# B&R Automation Studio project DynamicIO
Automation Studio 4.5.2.102

## Configuration 5AP1120

CPU 5PC901.TS77-00, AutomationRuntime D4.52, Build 4.1.2, Vc V4.52.0

### Task classes (Cpu.sw)
```
Cyclic#4:
  XmlConfigT <- Logic.XmlConfigTest.prg
  AsIoMManTe <- Logic.AsIoMManTest.prg
  ModuleIden <- Logic.ModuleIdent.prg [disabled]
Binaries: udbdef, TCData, ashwac, arconfig, asfw, ashwd, iomap, User, Role, sysconf
Libraries: standard, AsIOMMan, runtime, DataObj, AsXml, FileIO
```

### Hardware
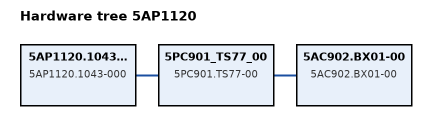
```
5AC902.BX01-00 : 5AC902.BX01-00 v1.1.1.0  [SY -> 5PC901_TS77_00.SY3]
5AP1120.1043-000 : 5AP1120.1043-000 v1.3.0.0
5PC901_TS77_00 : 5PC901.TS77-00 v2.0.0.0  [SY -> 5AP1120.1043-000.SY1]
  Connector IF1:
    AssignedOperatingSystem = ARemb
  Connector IF2:
    AssignedOperatingSystem = ARemb
  Connector IF3:
    AssignedOperatingSystem = ARemb
    ActivateDevice = 1
  Connector IF4:
    AssignedOperatingSystem = ARemb
    ActivateDevice = 1
  Connector IF5:
    AssignedOperatingSystem = ARemb
  Connector IF6:
    AssignedOperatingSystem = ARemb
  Connector IF7:
    AssignedOperatingSystem = ARemb
  Connector IF8:
    AssignedOperatingSystem = ARemb
  ConfigurationID = DynamicIO_5AP1120
  Simulation = 1
  FileDevice1
  FileDeviceName1 = root
  FileDevicePath1 = E:/
```

## Configuration CP3585

CPU X20CP3585, AutomationRuntime D4.52, Build 4.1.2, Vc V4.52.0

### Task classes (Cpu.sw)
```
Cyclic#3:
  XmlEditor <- Logic.XmlEditor.prg
Cyclic#4:
  IomapParse <- Logic.IomapParser.prg
  XmlConfigT <- Logic.XmlConfigTest.prg
  AsIoMManTe <- Logic.AsIoMManTest.prg
  ModuleIden <- Logic.ModuleIdent.prg
Binaries: udbdef, TCData, ashwac, arconfig, asfw, ashwd, iomap, User, Role, sysconf
Libraries: standard, AsIOMMan, runtime, DataObj, AsXml, FileIO, AsIODiag
```

### Hardware
```
X20BM11 : X20BM11 v1.0.0.1  [X2X1 -> X20CP3585.IF6]
X20CP3585 : X20CP3585 v1.5.0.0
  Connector IF2:
    ActivateDevice = 1
  ConfigurationID = DynamicIO_5AP1120
  Simulation = 1
  FileDevice1
  FileDeviceName1 = root
  FileDevicePath1 = E:/
X20DOF322 : X20DOF322 v1.1.2.0  [SS1 -> X20TB1F.SS; SL -> X20BM11.SL1]
X20TB1F : X20TB1F v1.0.0.0
```

## Logical view

Binary libraries used (declarations not repeated): operator, runtime, astime, AsIecCon, standard, AsIOMMan, DataObj, AsXml, FileIO, AsIODiag

### Global.typ - Global data types
```iecst
TYPE
	Module_type : 	STRUCT
		ModuleName : STRING[80];
		ModulePath : STRING[80];
		ChannelType : STRING[80] := 'BOOL';
		Channel : ARRAY[0..15]OF Channel_type;
		ModuleType : STRING[10] := '%QX';
	END_STRUCT;
	Channel_type : 	STRUCT
		ChannelVar : STRING[80];
		ChannelName : STRING[80];
	END_STRUCT;
END_TYPE
```

### Global.var - Global variables
```iecst
VAR
	X20DIF371 : Module_type;
	DI : ARRAY[0..15] OF BOOL;
	DigOut : ARRAY[0..15] OF BOOL;
	HW_config : Module_type;
	New_Variable : {REDUND_UNREPLICABLE} USINT := 4;
END_VAR
```


### Program Logical/Logic/ModuleIdent (ANSIC)

#### Types.typ
```iecst
TYPE
	ShowModules :
		(
		CONFIGURED_MODULES := 2,
		ALL := 3,
		PLUGGED := 1
		);
	ModuleInfo :
		(
		EPLAN_MODULE_TAG := 1007,
		HW_MODULE_NAME := 1006,
		PLUGGED_MODULE_BUS := 1004,
		CONFIGURATED_MODULE_BUS := 1005,
		PLUGGED_MODULE_NAME := 1002,
		CONFIG_MODULE_NAME := 1003,
		MODULE_PATH := 1001
		);
END_TYPE
```

#### Variables.var
```iecst
VAR
	GetInfo : DiagCreateInfo;
	Ident : UDINT;
	GetNumInfo : DiagGetNumInfo;
	GetStrInfo : DiagGetStrInfo;
	InfoDesc : STRING[80];
	start : BOOL;
	ConnectedModuleList : ARRAY[0..9] OF STRING[80];
	i : USINT;
END_VAR
```

#### Main.c
```c
#include <bur/plctypes.h>
#define TRUE	1
#define FALSE 	0

#ifdef _DEFAULT_INCLUDES
	#include <AsDefault.h>
#endif

void _INIT ProgramInit(void)
{

}

void _CYCLIC ProgramCyclic(void)
{
//	Тест опроса текущей конфигурации
	if(start)
	{
		if(GetInfo.ident == 0)	GetInfo.enable = TRUE;

		if(GetInfo.enable)
		{
			GetInfo.infoKind = CONFIGURED_MODULES;
			DiagCreateInfo(&GetInfo);
			Ident = GetInfo.ident;
			GetStrInfo.ident = Ident;
			GetStrInfo.enable = TRUE;
			GetStrInfo.infoCode = HW_MODULE_NAME;

			i = 0;
			if(GetInfo.status == 0)
			{
				GetInfo.enable = FALSE;
			}
		}
		if(	i < ( GetInfo.nrEntries) )
		{
			GetStrInfo.index = i;
			GetStrInfo.bufferLen = sizeof(InfoDesc);
			GetStrInfo.pBuffer = &InfoDesc;
			DiagGetStrInfo(&GetStrInfo);
			strcpy(ConnectedModuleList[GetStrInfo.index],InfoDesc);

			if(i == ( GetInfo.nrEntries - 1))
			{
				GetStrInfo.enable = FALSE;
				start = FALSE;
			}
			if(GetStrInfo.status == 0) i++;
		}
	}
}

void _EXIT ProgramExit(void)
{

}
```

### Program Logical/Logic/AsIoMManTest (ANSIC)

#### Types.typ
```iecst
TYPE
	FileMgrStep_enum :
		(
		CREATE,
		OPEN,
		WRITE,
		CLOSE
		);
	ReadCfg_enum :
		(
		Wait,
		CopyCfg,
		GetDatObjData,
		WriteXML
		);
END_TYPE
```

#### Variables.var
```iecst
VAR
	IOMMCopy : AsIOMMCopy;
	RemoveBr : AsIOMMRemove;
	CreateBr : AsIOMMCreate;
	status_message : STRING[128];
	error_string : STRING[128];
	step : USINT;
	error_status : UINT;
	error_step : USINT;
	error : BOOL;
	config : UINT;
	change_config : UINT;
	DataObjName : STRING[80];
	BR_ModuleName : STRING[80];
	DO_Create : DatObjCreate;
	DO_Read : DatObjRead;
	DO_Info : DatObjInfo;
	FileName : STRING[80];
	CfgReadStep : ReadCfg_enum;
	FW_Step : FileMgrStep_enum;
	Start : BOOL;
	fCreate : FileCreate;
	fOpen : FileOpen;
	fClose : FileClose;
	fRead : FileRead;
	fWrite : FileWrite;
	fIdent : UDINT;
END_VAR
```

#### Main.c
```c
#include <bur/plctypes.h>
#define	TRUE	1
#define	FALSE	0

#ifdef _DEFAULT_INCLUDES
	#include <AsDefault.h>
#endif

void _INIT ProgramInit(void)
{

}

void _CYCLIC ProgramCyclic(void)
{
	switch(CfgReadStep)
	{
		case Wait:
			if(Start)
			{
				CfgReadStep	= CopyCfg;
			}
			break;

		case CopyCfg:
			IOMMCopy.enable			= TRUE;
			IOMMCopy.pModuleName	= &BR_ModuleName;
			IOMMCopy.pNewModule		= &DataObjName;
			AsIOMMCopy(&IOMMCopy);
			if(IOMMCopy.status == ERR_OK)
			{
				CfgReadStep	= GetDatObjData;
			}
			break;

		case GetDatObjData:
			DO_Info.enable	= TRUE;
			DO_Info.pName	= IOMMCopy.pNewModule;
			DatObjInfo(&DO_Info);
			if(DO_Info.status == ERR_OK)
			{
				CfgReadStep	= WriteXML;
			}
			break;

		case WriteXML:
			switch (FW_Step)
			{

				case CREATE:
					fCreate.enable	= TRUE;
					fCreate.pDevice = (UDINT) "root";
					fCreate.pFile 	= &FileName;
					FileCreate(&fCreate);
					if(fCreate.status == ERR_OK)
					{
						fIdent	= fCreate.ident;
						FW_Step	= WRITE;
					}
					else if(fCreate.status == fiERR_EXIST)
					{
						FW_Step	= OPEN;
					}
					break;

				case OPEN:
					fOpen.pDevice	= (UDINT) "root";//= fCreate.pDevice;
					fOpen.pFile		= &FileName;//fCreate.pFile;
					fOpen.mode		= FILE_RW;
					fOpen.enable	= TRUE;
					FileOpen(&fOpen);
					if(fOpen.status == ERR_OK)
					{
						fIdent	= fOpen.ident;
						FW_Step	= WRITE;
					}
					break;

				case WRITE:
					fWrite.ident	= fIdent;
					fWrite.offset	= 0;
					fWrite.pSrc		= DO_Info.pDatObjMem;
					fWrite.len		= DO_Info.len;
					fWrite.enable	= TRUE;
					FileWrite(&fWrite);
					if(fWrite.status == ERR_OK)
					{
						FW_Step	= CLOSE;
					}
					break;

				case CLOSE:
					fClose.ident	= fIdent;
					fClose.enable	= TRUE;

					FileClose(&fClose);
					if(fClose.status == ERR_OK)
					{
						Start		= FALSE;
						CfgReadStep	= Wait;
					}
					break;

			}
	}
}

void _EXIT ProgramExit(void)
{

}
```

### Program Logical/Logic/XmlConfigTest (ANSIC)

#### Types.typ
```iecst
TYPE
	ProgramStep_enum :
		(
		Wait,
		WriteEndDoc,
		CreateMem,
		WriteArV,
		WriteHeader,
		WriteIO_Tag,
		WriteIO_TagAttr,
		WriteLinksTag,
		WriteLinkNodes,
		WriteLinksTagEnd,
		WriteIO_TagEnd,
		GetMemPointer,
		WriteDataObj,
		CopyXML,
		RemoveOldIomap,
		CreateNewIomap,
		DeleteDatObj,
		WarmRestart
		);
	FileMgrStep_enum :
		(
		CREATE,
		OPEN,
		WRITE,
		CLOSE
		);
	WriteLNStep_enum :
		(
		WriteLN_Tag,
		WriteLN_ID,
		WriteLN_Type,
		WriteProdTag,
		WriteProdDevice,
		WriteProdDPName,
		WriteProdKind,
		WriteProd_TagEnd,
		WriteConsTag,
		WriteConsDevice,
		WriteConsDPName,
		WriteConsKind,
		WriteCons_TagEnd,
		WriteLN_TagEnd
		);
	ModuleType : 	STRUCT
		ModuleName : STRING[80];
		ModulePath : STRING[80];
		ModuleType : STRING[80];
		ChanelNumber : USINT;
		ChanelType : STRING[80];
		ChanelVarName : ARRAY[0..15]OF STRING[80];
		ChanelName : ARRAY[0..15]OF STRING[80];
	END_STRUCT;
END_TYPE
```

#### Variables.var
```iecst
VAR
	CreateMemory : xmlCreateMemoryWriter;
	WriteStartDocument : xmlWriteStartDocument;
	WriteStartElement : xmlWriteStartElement;
	WriteAttribute : xmlWriteAttribute;
	WriteElementText : xmlWriteElementText;
	WriteEndElement : xmlWriteEndElement;
	WriteEndDocument : xmlWriteEndDocument;
	WritePI : xmlWritePI;
	GetMemoryInfo : xmlGetMemoryInfo;
	Step : ProgramStep_enum;
	Start : BOOL;
	XmlData : STRING[1000];
	Ident : UDINT;
	IO_AttrName : STRING[80] := 'xmlns';
	IOTagName : STRING[80] := 'IO';
	XmlEnc : STRING[80] := 'utf-8';
	fIdent : UDINT;
	XmlVer : STRING[80] := '1.0';
	IOAttrValue : STRING[80] := 'http://www.br-automation.com/AR/IO\';
	ArName : STRING[80] := 'AutomationRuntimeIOSystem';
	ArVer : STRING[80] := 'Version=\"1.0\"';
	fCreate : FileCreate;
	fOpen : FileOpen;
	fClose : FileClose;
	fRead : FileRead;
	LN_Step : WriteLNStep_enum;
	fWrite : FileWrite;
	FW_Step : FileMgrStep_enum;
	i : USINT := 5;
	DO_Delete : DatObjDelete;
	DO_Create : DatObjCreate;
	DO_Write : DatObjWrite;
	DO_Info : DatObjInfo;
	DataObj_Step : USINT;
	DOF322 : ModuleType;
	Buff : STRING[80];
	IOMMRemove : AsIOMMRemove;
	IOMMCreate : AsIOMMCreate;
END_VAR
```

#### Main.c
```c
#include <bur/plctypes.h>
#define TRUE	1
#define FALSE	0
UDINT StringCombiner(STRING* pDest,STRING* pIoType, STRING* pSrc1, STRING* pSrc2)
{
	strcpy(pDest,pIoType);
	strcat(pDest,".");
	strcat(pDest,pSrc1);
	strcat(pDest,".");
	strcat(pDest,pSrc2);
	return pDest;
}
#ifdef _DEFAULT_INCLUDES
	#include <AsDefault.h>
#endif

void _INIT ProgramInit(void)
{

	DigOut[1]	=	DigOut[1];
	DigOut[2]	=	DigOut[2];
	DigOut[3]	=	DigOut[3];
	DigOut[4]	=	DigOut[4];
	DigOut[5]	=	DigOut[5];
	DigOut[6]	=	DigOut[6];
	DigOut[7]	=	DigOut[7];
	DigOut[8]	=	DigOut[8];
	DigOut[9]	=	DigOut[9];
	DigOut[10]	=	DigOut[10];
	DigOut[11]	=	DigOut[11];
	DigOut[12]	=	DigOut[12];
	DigOut[13]	=	DigOut[13];
	DigOut[14]	=	DigOut[14];
	DigOut[15]	=	DigOut[15];

	Step	= Wait;
}

void _CYCLIC ProgramCyclic(void)
{
	switch(Step)
	{
		case Wait:
			if(Start)
			{
				strcpy(DOF322.ChanelName[0],"DigitalOutput01");
				strcpy(DOF322.ChanelName[1],"DigitalOutput02");
				strcpy(DOF322.ChanelName[2],"DigitalOutput03");
				strcpy(DOF322.ChanelName[3],"DigitalOutput04");
				strcpy(DOF322.ChanelName[4],"DigitalOutput05");
				strcpy(DOF322.ChanelName[5],"DigitalOutput06");
				strcpy(DOF322.ChanelName[6],"DigitalOutput07");
				strcpy(DOF322.ChanelName[7],"DigitalOutput08");
				strcpy(DOF322.ChanelName[8],"DigitalOutput09");
				strcpy(DOF322.ChanelName[9],"DigitalOutput10");
				strcpy(DOF322.ChanelName[10],"DigitalOutput11");
				strcpy(DOF322.ChanelName[11],"DigitalOutput12");
				strcpy(DOF322.ChanelName[12],"DigitalOutput13");
				strcpy(DOF322.ChanelName[13],"DigitalOutput14");
				strcpy(DOF322.ChanelName[14],"DigitalOutput15");
				strcpy(DOF322.ChanelName[15],"DigitalOutput16");

				strcpy(DOF322.ChanelVarName[0],"::DigOut[15]");
				strcpy(DOF322.ChanelVarName[1],"::DigOut[14]");
				strcpy(DOF322.ChanelVarName[2],"::DigOut[13]");
				strcpy(DOF322.ChanelVarName[3],"::DigOut[12]");
				strcpy(DOF322.ChanelVarName[4],"::DigOut[11]");
				strcpy(DOF322.ChanelVarName[5],"::DigOut[10]");
				strcpy(DOF322.ChanelVarName[6],"::DigOut[9]");
				strcpy(DOF322.ChanelVarName[7],"::DigOut[8]");
				strcpy(DOF322.ChanelVarName[8],"::DigOut[7]");
				strcpy(DOF322.ChanelVarName[9],"::DigOut[6]");
				strcpy(DOF322.ChanelVarName[10],"::DigOut[5]");
				strcpy(DOF322.ChanelVarName[11],"::DigOut[4]");
				strcpy(DOF322.ChanelVarName[12],"::DigOut[3]");
				strcpy(DOF322.ChanelVarName[13],"::DigOut[2]");
				strcpy(DOF322.ChanelVarName[14],"::DigOut[1]");
				strcpy(DOF322.ChanelVarName[15],"::DigOut[0]");

				strcpy(DOF322.ChanelType,"BOOL");
				strcpy(DOF322.ModulePath,"SL1.IF2.ST3");
				strcpy(DOF322.ModuleName,"SL1.IF2.ST3");
				Step	= CreateMem;
			}
			break;

		case CreateMem:
			CreateMemory.enable		= TRUE;
			xmlCreateMemoryWriter(&CreateMemory);
			if( CreateMemory.status == ERR_OK )
			{
				Ident	= CreateMemory.ident;
				Step	= WriteHeader;
			}
			break;

		case WriteHeader:
			WriteStartDocument.ident		= Ident;
			WriteStartDocument.enable		= TRUE;
		//	WriteStartDocument.pEncoding	= &XmlEnc;
			WriteStartDocument.pVersion		= (UDINT) "1.0";
			xmlWriteStartDocument(&WriteStartDocument);
			if(WriteStartDocument.status == ERR_OK)
			{
				Step	= WriteArV;
			}

			break;
		case WriteArV:
			WritePI.ident	= Ident;
			WritePI.pTarget	= (UDINT) "AutomationRuntimeIOSystem";
			WritePI.pValue	= (UDINT) "Version=\"1.0\"";
			WritePI.enable	= TRUE;
			xmlWritePI(&WritePI);
			if(WritePI.status == ERR_OK)
			{
				Step	= WriteIO_Tag;
			}

			break;

		case WriteIO_Tag:
			WriteStartElement.ident		= Ident;
			WriteStartElement.pName		= (UDINT) "IO";
			WriteStartElement.enable	= TRUE;
			xmlWriteStartElement(&WriteStartElement);
			if(WriteStartElement.status == ERR_OK)
			{
				Step = WriteIO_TagAttr;
			}

			break;

		case WriteIO_TagAttr:
			WriteAttribute.ident	= Ident;
			WriteAttribute.pName	= (UDINT) "xmlns";
			WriteAttribute.pValue	= (UDINT) "http://www.br-automation.com/AR/IO";
			WriteAttribute.enable	= TRUE;
			xmlWriteAttribute(&WriteAttribute);
			if(WriteAttribute.status == ERR_OK)
			{
				Step	= WriteLinksTag;
			}
			break;

		case WriteLinksTag:
			WriteStartElement.ident		= Ident;
			WriteStartElement.pName		= (UDINT) "Links";
			WriteStartElement.enable	= TRUE;
			xmlWriteStartElement(&WriteStartElement);
			if(WriteStartElement.status == ERR_OK)
			{
				WriteStartElement.enable	= 0;
				Step = WriteLinkNodes;
				LN_Step	= WriteLN_Tag;
				i = 0;
			}

			break;

		case WriteLinkNodes:

			switch(LN_Step)
			{
				case WriteLN_Tag:
					WriteStartElement.ident		= Ident;
					WriteStartElement.pName		= (UDINT) "LN";
					WriteStartElement.enable	= TRUE;
					xmlWriteStartElement(&WriteStartElement);
					if(WriteStartElement.status == ERR_OK)
					{
						LN_Step = WriteLN_ID;
					}

					break;

				case WriteLN_ID:
				//STRING Buff[80];
					WriteAttribute.ident	= Ident;
					WriteAttribute.pName	= (UDINT) "ID";
					WriteAttribute.pValue	= (UDINT) StringCombiner(&Buff,"%QX",DOF322.ModulePath,DOF322.ChanelName[i]);/*"SL1.IF2.ST1.SL1.Input01"*/
					WriteAttribute.enable	= TRUE;
					xmlWriteAttribute(&WriteAttribute);
					if(WriteAttribute.status == ERR_OK)
					{
						LN_Step	= WriteLN_Type;
					}
					break;

				case WriteLN_Type:
					WriteAttribute.ident	= Ident;
					WriteAttribute.pName	= (UDINT) "Type";
					WriteAttribute.pValue	= &DOF322.ChanelType; //(UDINT) "BOOL";
					WriteAttribute.enable	= TRUE;
					xmlWriteAttribute(&WriteAttribute);
					if(WriteAttribute.status == ERR_OK)
					{
						LN_Step	= WriteProdTag;
					}
					break;

				case WriteProdTag:
					WriteStartElement.ident		= Ident;
					WriteStartElement.pName		= (UDINT) "Prod";
					WriteStartElement.enable	= TRUE;
					xmlWriteStartElement(&WriteStartElement);
					if(WriteStartElement.status == ERR_OK)
					{
						LN_Step = WriteProdDevice;
					}

					break;

				case WriteProdDevice:
					WriteAttribute.ident	= Ident;
					WriteAttribute.pName	= (UDINT) "Device";
					WriteAttribute.pValue	= &DOF322.ModulePath; //(UDINT) "SL1.IF2.ST1.SL2";
					WriteAttribute.enable	= TRUE;
					xmlWriteAttribute(&WriteAttribute);
					if(WriteAttribute.status == ERR_OK)
					{
						WriteAttribute.enable	= FALSE;
						LN_Step	= WriteProdDPName;
					}
					break;

				case WriteProdDPName:
					WriteAttribute.ident	= Ident;
					WriteAttribute.pName	= (UDINT) "DPName";
					WriteAttribute.pValue	= &DOF322.ChanelName[i]; //(UDINT) "Input01";
					WriteAttribute.enable	= TRUE;
					xmlWriteAttribute(&WriteAttribute);
					if(WriteAttribute.status == ERR_OK)
					{
						LN_Step	= WriteProdKind;
						WriteAttribute.enable	= FALSE;
					}
					break;

				case WriteProdKind:
					WriteAttribute.ident	= Ident;
					WriteAttribute.pName	= (UDINT) "Kind";
					WriteAttribute.pValue	= (UDINT) "io";
					WriteAttribute.enable	= TRUE;
					xmlWriteAttribute(&WriteAttribute);
					if(WriteAttribute.status == ERR_OK)
					{
						WriteAttribute.enable	= FALSE;
						LN_Step	= WriteProd_TagEnd;
					}
					break;
				case WriteProd_TagEnd:
					WriteEndElement.ident	= Ident;
					WriteEndElement.enable	= TRUE;
					xmlWriteEndElement(&WriteEndElement);
					if(WriteEndElement.status	== ERR_OK)
					{
						LN_Step	= WriteConsTag;
						WriteEndElement.enable	= FALSE;
						WriteStartElement.enable	= FALSE;
					}
					break;

				case WriteConsTag:
					WriteStartElement.ident		= Ident;
					WriteStartElement.pName		= (UDINT) "Cons";
					WriteStartElement.enable	= TRUE;
					xmlWriteStartElement(&WriteStartElement);
					if(WriteStartElement.status == ERR_OK)
					{
						LN_Step = WriteConsDevice;
					}

					break;

				case WriteConsDevice:
					WriteAttribute.ident	= Ident;
					WriteAttribute.pName	= (UDINT) "Device";
					WriteAttribute.pValue	= (UDINT) "TC#1-CPYDEV";
					WriteAttribute.enable	= TRUE;
					xmlWriteAttribute(&WriteAttribute);
					if(WriteAttribute.status == ERR_OK)
					{
						LN_Step	= WriteConsDPName;
					}
					break;

				case WriteConsDPName:
					WriteAttribute.ident	= Ident;
					WriteAttribute.pName	= (UDINT) "DPName";
					WriteAttribute.pValue	= &DOF322.ChanelVarName[i];
					WriteAttribute.enable	= TRUE;
					xmlWriteAttribute(&WriteAttribute);
					if(WriteAttribute.status == ERR_OK)
					{
						LN_Step	= WriteConsKind;
					}
					break;

				case WriteConsKind:
					WriteAttribute.ident	= Ident;
					WriteAttribute.pName	= (UDINT) "Kind";
					WriteAttribute.pValue	= (UDINT) "pv";
					WriteAttribute.enable	= TRUE;
					xmlWriteAttribute(&WriteAttribute);
					if(WriteAttribute.status == ERR_OK)
					{
						LN_Step	= WriteCons_TagEnd;
					}
					break;

				case WriteCons_TagEnd:
					WriteEndElement.ident	= Ident;
					WriteEndElement.enable	= TRUE;
					xmlWriteEndElement(&WriteEndElement);
					if(WriteEndElement.status	== ERR_OK)
					{
						LN_Step	= WriteLN_TagEnd;
					}
					break;

				case WriteLN_TagEnd:
					WriteEndElement.ident	= Ident;
					WriteEndElement.enable	= TRUE;
					xmlWriteEndElement(&WriteEndElement);
					if(WriteEndElement.status	== ERR_OK)
					{
						i++;
						if(i<DOF322.ChanelNumber)
							{

								LN_Step	= WriteLN_Tag;

							}
							else
							{
								Step	= WriteLinksTagEnd;
							}
					}
					break;

			}
			break;

		case WriteLinksTagEnd:
			WriteEndElement.ident	= Ident;
			WriteEndElement.enable	= TRUE;
			xmlWriteEndElement(&WriteEndElement);
			if(WriteEndElement.status	== ERR_OK)
			{

				Step	= WriteIO_TagEnd;
			}
			break;

		case WriteIO_TagEnd:
			WriteEndElement.ident	= Ident;
			WriteEndElement.enable	= TRUE;
			xmlWriteEndElement(&WriteEndElement);
			if(WriteEndElement.status	== ERR_OK)
			{
				Step	= WriteEndDoc;
			}
			break;

		case WriteEndDoc:
			WriteEndDocument.ident	= Ident;
			WriteEndDocument.enable	= TRUE;
			xmlWriteEndDocument(&WriteEndDocument);
			if(WriteEndDocument.status	== ERR_OK)
			{
				Step	= GetMemPointer;
			}
			break;

		case GetMemPointer:
			GetMemoryInfo.ident		= Ident;
			GetMemoryInfo.enable	= TRUE;
			xmlGetMemoryInfo(&GetMemoryInfo);
			if(GetMemoryInfo.status	== ERR_OK)
			{
				Step	= WriteDataObj;
				FW_Step	= OPEN;
			}
			break;

		case WriteDataObj:
			DO_Create.enable	= TRUE;
			DO_Create.pName		= (UDINT)	"NewIomap";
			DO_Create.MemType	= doTEMP;
			DO_Create.pCpyData	= GetMemoryInfo.pXmlData;
			DO_Create.len		= GetMemoryInfo.xmlDataSize;
			DatObjCreate(&DO_Create);
			if(DO_Create.status == ERR_OK)
			{
				Step = CopyXML;
			}
			break;

		case CopyXML:
			//memcpy(&XmlData,GetMemoryInfo.pXmlData,GetMemoryInfo.xmlDataSize);
			switch (FW_Step)
			{
			/*
			case CREATE:
					fCreate.enable = TRUE;
					fCreate.pDevice = (UDINT) "root";
					fCreate.pFile = (UDINT) "test.xml";
					FileCreate(&fCreate);
					if(fCreate.status == ERR_OK)
					{
						fIdent	= fCreate.ident;
						step	= WRITE;
					}
					break;
			*/
			case OPEN:
					fOpen.pDevice	=	(UDINT) "root";//= fCreate.pDevice;
					fOpen.pFile	= (UDINT) "test.xml";//fCreate.pFile;
					fOpen.mode	= FILE_RW;
				fOpen.enable	= TRUE;
				FileOpen(&fOpen);
				if(fOpen.status == ERR_OK)
				{
					fIdent	= fOpen.ident;
					FW_Step	= WRITE;
				}
				break;

			case WRITE:
				fWrite.ident	= fIdent;
				fWrite.offset	= 0;
				fWrite.pSrc		= GetMemoryInfo.pXmlData;//DO_Create.pDatObjMem;
				fWrite.len		= GetMemoryInfo.xmlDataSize;//DO_Create.len;
				fWrite.enable	= TRUE;
				FileWrite(&fWrite);
				if(fWrite.status == ERR_OK)
				{
					FW_Step	= CLOSE;
				}
				break;

			case CLOSE:
				fClose.ident	= fIdent;
				fClose.enable	= TRUE;

				FileClose(&fClose);
				if(fClose.status == ERR_OK)
				{
					//Start	= FALSE;
					Step	= RemoveOldIomap;
				}
				break;

			}

			break;

		case RemoveOldIomap:
			IOMMRemove.enable	= TRUE;
			IOMMRemove.pModuleName = (UDINT) "iomap";
			AsIOMMRemove(&IOMMRemove);
			if(IOMMRemove.status == ERR_OK)
			{
				Step	= CreateNewIomap;
			}
			else if(IOMMRemove.status == iommERR_NOSUCH_MODULE)
			{
				Step	= CreateNewIomap;
			}
			break;

		case CreateNewIomap:
			IOMMCreate.enable	= TRUE;
			IOMMCreate.pDataObject	=  DO_Create.pName;
			IOMMCreate.memType		= doUSRROM;
			IOMMCreate.moduleKind	= iommMAPPING;
			IOMMCreate.pNewModule	= (UDINT) "iomap";
			AsIOMMCreate(&IOMMCreate);
			if(IOMMCreate.status == ERR_OK)
			{
				Step	= DeleteDatObj;//DeleteDatObj;
			}
			break;

		case DeleteDatObj:
			DO_Delete.enable	= TRUE;
			DO_Delete.ident		= DO_Create.ident;
			DatObjDelete(&DO_Delete);
			if(DO_Delete.status == ERR_OK)
			{
				Step	= WarmRestart;
			}
			break;

		case WarmRestart:
			Start	= FALSE;
			Step	= Wait;
			break;

	}
}

void _EXIT ProgramExit(void)
{

}
```

### Program Logical/Logic/XmlEditor (ANSIC)

#### Types.typ
```iecst
TYPE
	FileMgrStep_enum :
		(
		CREATE,
		OPEN,
		WRITE,
		CLOSE
		);
	ReadCfg_enum :
		(
		Wait,
		CopyCfg,
		GetDatObjData,
		CreateMemReader,
		ReadXmlNode,
		ReadXmlNodeAttributes,
		DeleteDataObject,
		WriteXML,
		CloseMemReader
		);
	XmlNode_type : 	STRUCT
		NodeName : STRING[80];
		NodeValue : STRING[80];
		NodeAttr : ARRAY[0..14]OF XmlNodeAttr_type;
	END_STRUCT;
	XmlNodeAttr_type : 	STRUCT
		AttrName : STRING[80];
		AttrValue : STRING[80];
	END_STRUCT;
END_TYPE
```

#### Variables.var
```iecst
VAR
	IOMMCopy : AsIOMMCopy;
	DataObjName : STRING[80];
	BR_ModuleName : STRING[80];
	DO_Create : DatObjCreate;
	DO_Read : DatObjRead;
	DO_Delete : DatObjDelete;
	DO_Info : DatObjInfo;
	FileName : STRING[80];
	CfgReadStep : ReadCfg_enum;
	FW_Step : FileMgrStep_enum;
	Start : BOOL;
	fCreate : FileCreate;
	fOpen : FileOpen;
	fClose : FileClose;
	fRead : FileRead;
	fWrite : FileWrite;
	fIdent : UDINT;
	Buff : STRING[80];
	CreateMemoryReader : xmlCreateMemoryReader;
	ReadNextNode : xmlReadNextNode;
	ReadAttributeNr : xmlReadAttributeNr;
	NodeName : STRING[80];
	NodeValue : STRING[80];
	XmlNode : ARRAY[0..254] OF XmlNode_type;
	attrNr : USINT;
	NodeNr : USINT;
	CloseMemoryReader : xmlCloseMemoryReader;
END_VAR
```

#### Main.c
```c
#include <bur/plctypes.h>
#define TRUE	1
#define	FALSE	0
#ifdef _DEFAULT_INCLUDES
	#include <AsDefault.h>
#endif

void _INIT ProgramInit(void)
{

}

void _CYCLIC ProgramCyclic(void)
{

	switch(CfgReadStep)
	{
		case Wait:
			if(Start)
			{
				CfgReadStep	= CopyCfg;
			}
			break;

		case CopyCfg:
			IOMMCopy.enable			= TRUE;
			IOMMCopy.pModuleName	= &BR_ModuleName;
			IOMMCopy.pNewModule		= &DataObjName;
			IOMMCopy.memType		= doTEMP;
			AsIOMMCopy(&IOMMCopy);
			if(IOMMCopy.status == ERR_OK)
			{
				CfgReadStep			= GetDatObjData;
			}
			break;

		case GetDatObjData:
			DO_Info.enable	= TRUE;
			DO_Info.pName	= IOMMCopy.pNewModule;
			DatObjInfo(&DO_Info);
			if(DO_Info.status == ERR_OK)
			{
				CfgReadStep	= CreateMemReader;
			}
			break;

		case CreateMemReader:
			CreateMemoryReader.enable		= TRUE;
			CreateMemoryReader.pXmlMemory	= DO_Info.pDatObjMem;
			CreateMemoryReader.memorySize	= DO_Info.len;
			xmlCreateMemoryReader(&CreateMemoryReader);
			if(CreateMemoryReader.status == ERR_OK)
			{
				CfgReadStep			= ReadXmlNode;
				NodeNr 				= 0;
				ReadNextNode.enable	= TRUE;
			}
			break;

		case ReadXmlNode:
			ReadNextNode.ident		= CreateMemoryReader.ident;
			ReadNextNode.pName		= (UDINT) &XmlNode[NodeNr].NodeName;
			ReadNextNode.nameSize	= sizeof(XmlNode[NodeNr].NodeName);
			ReadNextNode.pValue		= (UDINT) &XmlNode[NodeNr].NodeValue;
			ReadNextNode.valueSize	= sizeof(XmlNode[NodeNr].NodeValue);
			xmlReadNextNode(&ReadNextNode);
			if(NodeNr>253)
			{
				CfgReadStep	= WriteXML;
			}
			else if(ReadNextNode.status == ERR_OK)
			{
				attrNr				= 0;
				ReadNextNode.enable	= FALSE;
				CfgReadStep			= ReadXmlNodeAttributes;
			}
			else if(ReadNextNode.status == xmlERR_NO_FURTHER_XML_NODE)
			{
				CfgReadStep	= WriteXML;
			}

			break;

		case ReadXmlNodeAttributes:
			if(attrNr < ReadNextNode.attributeCount)
			{
				ReadAttributeNr.ident		= ReadNextNode.ident;
				ReadAttributeNr.enable		= TRUE;
				ReadAttributeNr.index		= attrNr;
				ReadAttributeNr.pName		= (UDINT) &XmlNode[NodeNr].NodeAttr[attrNr].AttrName;
				ReadAttributeNr.nameSize	= sizeof(XmlNode[NodeNr].NodeAttr[attrNr].AttrName);
				ReadAttributeNr.pValue		= (UDINT) &XmlNode[NodeNr].NodeAttr[attrNr].AttrValue;
				ReadAttributeNr.valueSize	= sizeof(XmlNode[NodeNr].NodeAttr[attrNr].AttrValue);
				xmlReadAttributeNr(&ReadAttributeNr);
				if(ReadAttributeNr.status	==	ERR_OK)
				{
					attrNr++;
				}

			}
			else
			{
				NodeNr++;
				ReadNextNode.enable	= TRUE;
				CfgReadStep			= ReadXmlNode;
			}
			break;

		case WriteXML:
			switch (FW_Step)
			{

				case CREATE:
					fCreate.enable	= TRUE;
					fCreate.pDevice = (UDINT) "root";
					fCreate.pFile	= &FileName;
					FileCreate(&fCreate);
					if(fCreate.status == ERR_OK)
					{
						fIdent	= fCreate.ident;
						FW_Step	= WRITE;
					}
					else if(fCreate.status == fiERR_EXIST)
					{
						FW_Step	= OPEN;
					}
					break;

				case OPEN:
					fOpen.pDevice	=	(UDINT) "root";//= fCreate.pDevice;
					fOpen.pFile		= &FileName;//fCreate.pFile;
					fOpen.mode		= FILE_RW;
					fOpen.enable	= TRUE;
					FileOpen(&fOpen);
					if(fOpen.status == ERR_OK)
					{
						fIdent	= fOpen.ident;
						FW_Step	= WRITE;
					}
					break;

				case WRITE:
					fWrite.ident	= fIdent;
					fWrite.offset	= 0;
					fWrite.pSrc		= DO_Info.pDatObjMem;
					fWrite.len		= DO_Info.len;
					fWrite.enable	= TRUE;
					FileWrite(&fWrite);
					if(fWrite.status == ERR_OK)
					{
						FW_Step	= CLOSE;
					}
					break;

				case CLOSE:
					fClose.ident	= fIdent;
					fClose.enable	= TRUE;
					FileClose(&fClose);
					if(fClose.status == ERR_OK)
					{
						CfgReadStep	= DeleteDataObject;
					}
					break;
			}
			break;

		case DeleteDataObject:
			DO_Delete.enable	= TRUE;
			DO_Delete.ident		= DO_Info.ident;
			DatObjDelete(&DO_Delete);
			if(DO_Delete.status == ERR_OK)
			{
				CfgReadStep	= CloseMemReader;
			}
			break;

		case CloseMemReader:
			CloseMemoryReader.enable	= TRUE;
			CloseMemoryReader.ident		= CreateMemoryReader.ident;
			xmlCloseMemoryReader(&CloseMemoryReader);
			if(CloseMemoryReader.status == ERR_OK)
			{
				CfgReadStep	= Wait;
				Start		= FALSE;
			}
			break;

	}

}

void _EXIT ProgramExit(void)
{

}
```

### Program Logical/Logic/IomapParser (ANSIC)

#### Types.typ
```iecst
TYPE
	FileMgrStep_enum :
		(
		CREATE,
		OPEN,
		WRITE,
		CLOSE
		);
	ReadCfg_enum :
		(
		WAIT,
		READ_HW_CONFIG,
		COPY_CFG,
		GET_DATOBJ_INFO,
		CREATE_MEM_READER,
		READ_NEXT_NODE,
		READ_LN_ATTR,
		READ_PROD_ATTR,
		READ_CONS_ATTR,
		WRITE_XML,
		DELETE_DAT_OBJ,
		CLOSE_MEM_READER,
		ERROR
		);
	XmlNode_type : 	STRUCT
		NodeName : STRING[80];
		NodeValue : STRING[80];
		NodeAttr : XmlNodeAttr_type;
	END_STRUCT;
	XmlNodeAttr_type : 	STRUCT
		AttrName : STRING[80];
		AttrValue : STRING[80];
	END_STRUCT;
	LN_type : 	STRUCT
		ID : STRING[80];
		Type : STRING[80];
		Prod : Prod_type;
		Cons : Cons_type;
	END_STRUCT;
	Cons_type : 	STRUCT
		Device : STRING[80];
		DPName : STRING[80];
		Kind : STRING[10];
	END_STRUCT;
	Prod_type : 	STRUCT
		Device : STRING[80];
		DPName : STRING[80];
		Kind : STRING[10];
	END_STRUCT;
END_TYPE
```

#### Variables.var
```iecst
VAR
	IOMMCopy : AsIOMMCopy;
	DataObjName : STRING[80];
	BR_ModuleName : STRING[80];
	DO_Create : DatObjCreate;
	DO_Read : DatObjRead;
	DO_Delete : DatObjDelete;
	DO_Info : DatObjInfo;
	FileName : STRING[80];
	CfgReadStep : ReadCfg_enum;
	FW_Step : FileMgrStep_enum;
	Start : BOOL;
	fCreate : FileCreate;
	fOpen : FileOpen;
	fClose : FileClose;
	fRead : FileRead;
	fWrite : FileWrite;
	fIdent : UDINT;
	Buff : STRING[80];
	CreateMemoryReader : xmlCreateMemoryReader;
	ReadNextNode : xmlReadNextNode;
	ReadAttributeNr : xmlReadAttributeNr;
	NodeName : STRING[80];
	NodeValue : STRING[80];
	XmlNode : XmlNode_type;
	attrNr : USINT;
	NodeNr : USINT;
	CloseMemoryReader : xmlCloseMemoryReader;
	LinkNode : LN_type;
END_VAR
```

#### Main.c
```c
#include <bur/plctypes.h>
#define TRUE	1
#define	FALSE	0
#ifdef _DEFAULT_INCLUDES
	#include <AsDefault.h>
#endif

void _INIT ProgramInit(void)
{
	Start		= FALSE;
	CfgReadStep	= WAIT;
}

void _CYCLIC ProgramCyclic(void)
{

	switch(CfgReadStep)
	{
		case WAIT:
			if(Start)
			{
				CfgReadStep	= COPY_CFG;
			}
			break;

		/*case READ_HW_CONFIG:
			if(GetInfo.ident == 0)	GetInfo.enable = TRUE;

			if(GetInfo.enable)
			{
				GetInfo.infoKind = CONFIGURED_MODULES;
				DiagCreateInfo(&GetInfo);
				Ident = GetInfo.ident;
				GetStrInfo.ident = Ident;
				GetStrInfo.enable = TRUE;
				GetStrInfo.infoCode = HW_MODULE_NAME;

				i = 0;
				if(GetInfo.status == 0)
				{
					GetInfo.enable = FALSE;
				}
			}
			if(	i < ( GetInfo.nrEntries) )
			{
				GetStrInfo.index = i;
				GetStrInfo.bufferLen = sizeof(InfoDesc);
				GetStrInfo.pBuffer = &InfoDesc;
				DiagGetStrInfo(&GetStrInfo);
				strcpy(ConnectedModuleList[GetStrInfo.index],InfoDesc);

				if(i == ( GetInfo.nrEntries - 1))
				{
					GetStrInfo.enable = FALSE;
					start = FALSE;
				}
				if(GetStrInfo.status == 0) i++;
			}
			break;
		*/
		case COPY_CFG:
			IOMMCopy.enable			= TRUE;
			IOMMCopy.pModuleName	= (UDINT) "iomap";//&BR_ModuleName;
			IOMMCopy.pNewModule		= (UDINT) "temp";
			IOMMCopy.memType		= doTEMP;

			AsIOMMCopy(&IOMMCopy);

			if(IOMMCopy.status == ERR_OK)
			{
				CfgReadStep	= GET_DATOBJ_INFO;
			}
			break;

		case GET_DATOBJ_INFO:
			DO_Info.enable	= TRUE;
			DO_Info.pName	= IOMMCopy.pNewModule;

			DatObjInfo(&DO_Info);

			if(DO_Info.status == ERR_OK)
			{
				CfgReadStep	= CREATE_MEM_READER;
			}
			break;

		case CREATE_MEM_READER:
			CreateMemoryReader.enable		= TRUE;
			CreateMemoryReader.pXmlMemory	= DO_Info.pDatObjMem;
			CreateMemoryReader.memorySize	= DO_Info.len;

			xmlCreateMemoryReader(&CreateMemoryReader);

			if(CreateMemoryReader.status == ERR_OK)
			{
				CfgReadStep	= READ_NEXT_NODE;

			}
			break;

		case READ_NEXT_NODE:
			ReadNextNode.ident		= CreateMemoryReader.ident;
			ReadNextNode.pName		= (UDINT) &XmlNode.NodeName;
			ReadNextNode.nameSize	= sizeof(XmlNode.NodeName);
			ReadNextNode.pValue		= (UDINT) &XmlNode.NodeValue;
			ReadNextNode.valueSize	= sizeof(XmlNode.NodeValue);

			xmlReadNextNode(&ReadNextNode);

			if(ReadNextNode.status == ERR_OK)
			{
				if( (strcmp(&XmlNode.NodeName,(UDINT) "LN") == 0 ) && ( ReadNextNode.attributeCount != 0 ) )
				{
					CfgReadStep	= READ_LN_ATTR;
				}
				else if( (strcmp(&XmlNode.NodeName,(UDINT) "Prod") == 0 ) && ( ReadNextNode.attributeCount != 0 ) )
				{
					CfgReadStep	= READ_PROD_ATTR;
				}
				else if( (strcmp(&XmlNode.NodeName,(UDINT) "Cons") == 0 ) && ( ReadNextNode.attributeCount != 0 ) )
				{
					CfgReadStep	= READ_CONS_ATTR;
				}
				else
				{
					CfgReadStep	= READ_NEXT_NODE;
				}
			}
			else if(ReadNextNode.status == xmlERR_NO_FURTHER_XML_NODE)
			{
				CfgReadStep	= DELETE_DAT_OBJ;
			}

			break;

		case READ_LN_ATTR:
			if(attrNr < ReadNextNode.attributeCount)
			{
				ReadAttributeNr.enable		= TRUE;
				ReadAttributeNr.ident		= ReadNextNode.ident;
				ReadAttributeNr.index		= attrNr;
				ReadAttributeNr.pName		= (UDINT) &XmlNode.NodeAttr.AttrName;
				ReadAttributeNr.nameSize	= sizeof(XmlNode.NodeAttr.AttrName);
				ReadAttributeNr.pValue		= (UDINT) &XmlNode.NodeAttr.AttrValue;
				ReadAttributeNr.valueSize	= sizeof(XmlNode.NodeAttr.AttrValue);

				xmlReadAttributeNr(&ReadAttributeNr);

				if(ReadAttributeNr.status	==	ERR_OK)
				{
					if( strcmp(&XmlNode.NodeAttr.AttrName,(UDINT) "ID") == 0 )
					{
						strcpy(LinkNode.ID,XmlNode.NodeAttr.AttrValue);
					}
					else if( strcmp(&XmlNode.NodeAttr.AttrName,(UDINT) "Type") == 0 )
					{
						strcpy(LinkNode.Type,XmlNode.NodeAttr.AttrValue);
					}

					attrNr++;
				}

			}
			else
			{
				attrNr		= 0;
				CfgReadStep	= READ_NEXT_NODE;
			}
			break;

		case READ_PROD_ATTR:
			if(attrNr < ReadNextNode.attributeCount)
			{
				ReadAttributeNr.enable		=	TRUE;
				ReadAttributeNr.ident		= ReadNextNode.ident;
				ReadAttributeNr.index		= attrNr;
				ReadAttributeNr.pName		= (UDINT) &XmlNode.NodeAttr.AttrName;
				ReadAttributeNr.nameSize	= sizeof(XmlNode.NodeAttr.AttrName);
				ReadAttributeNr.pValue		= (UDINT) &XmlNode.NodeAttr.AttrValue;
				ReadAttributeNr.valueSize	= sizeof(XmlNode.NodeAttr.AttrValue);

				xmlReadAttributeNr(&ReadAttributeNr);

				if(ReadAttributeNr.status	==	ERR_OK)
				{
					if( strcmp(&XmlNode.NodeAttr.AttrName,(UDINT) "Device") == 0 )
					{
						strcpy(LinkNode.Prod.Device,XmlNode.NodeAttr.AttrValue);
					}
					else if( strcmp(&XmlNode.NodeAttr.AttrName,(UDINT) "DPName") == 0 )
					{
						strcpy(LinkNode.Prod.DPName,XmlNode.NodeAttr.AttrValue);
					}
					else if( strcmp(&XmlNode.NodeAttr.AttrName,(UDINT) "Kind") == 0 )
					{
						strcpy(LinkNode.Prod.Kind,XmlNode.NodeAttr.AttrValue);
					}

					attrNr++;
				}
			}
			else
			{
				attrNr		= 0;
				CfgReadStep	= READ_NEXT_NODE;
			}
			break;

		case READ_CONS_ATTR:
			if( attrNr < ReadNextNode.attributeCount )
			{
				ReadAttributeNr.enable		= TRUE;
				ReadAttributeNr.ident		= ReadNextNode.ident;
				ReadAttributeNr.index		= attrNr;
				ReadAttributeNr.pName		= (UDINT) &XmlNode.NodeAttr.AttrName;
				ReadAttributeNr.nameSize	= sizeof(XmlNode.NodeAttr.AttrName);
				ReadAttributeNr.pValue		= (UDINT) &XmlNode.NodeAttr.AttrValue;
				ReadAttributeNr.valueSize	= sizeof(XmlNode.NodeAttr.AttrValue);

				xmlReadAttributeNr(&ReadAttributeNr);

				if(ReadAttributeNr.status	==	ERR_OK)
				{
					if( strcmp(&XmlNode.NodeAttr.AttrName,(UDINT) "Device") == 0 )
					{
						strcpy(LinkNode.Cons.Device,XmlNode.NodeAttr.AttrValue);
					}
					else if( strcmp(&XmlNode.NodeAttr.AttrName,(UDINT) "DPName") == 0 )
					{
						strcpy(LinkNode.Cons.DPName,XmlNode.NodeAttr.AttrValue);
					}
					else if( strcmp(&XmlNode.NodeAttr.AttrName,(UDINT) "Kind") == 0 )
					{
						strcpy(LinkNode.Cons.Kind,XmlNode.NodeAttr.AttrValue);
					}

					attrNr++;
				}
			}
			else
			{
				attrNr		= 0;
				CfgReadStep	= READ_NEXT_NODE;
			}
			break;

		case WRITE_XML:
			switch (FW_Step)
			{

				case CREATE:
					fCreate.enable	= TRUE;
					fCreate.pDevice	= (UDINT) "root";
					fCreate.pFile	= &FileName;

					FileCreate(&fCreate);

					if(fCreate.status == ERR_OK)
					{
						fIdent	= fCreate.ident;
						FW_Step	= WRITE;
					}
					else if(fCreate.status == fiERR_EXIST)
					{
						FW_Step	= OPEN;
					}
					break;

				case OPEN:
					fOpen.pDevice	=	(UDINT) "root";//= fCreate.pDevice;
					fOpen.pFile		= &FileName;//fCreate.pFile;
					fOpen.mode		= FILE_RW;
					fOpen.enable	= TRUE;

					FileOpen(&fOpen);

					if(fOpen.status == ERR_OK)
					{
						fIdent	= fOpen.ident;
						FW_Step	= WRITE;
					}
					break;

				case WRITE:
					fWrite.ident	= fIdent;
					fWrite.offset	= 0;
					fWrite.pSrc		= DO_Info.pDatObjMem;
					fWrite.len		= DO_Info.len;
					fWrite.enable	= TRUE;

					FileWrite(&fWrite);

					if(fWrite.status == ERR_OK)
					{
						FW_Step	= CLOSE;
					}
					break;

				case CLOSE:
					fClose.ident	= fIdent;
					fClose.enable	= TRUE;

					FileClose(&fClose);

					if(fClose.status == ERR_OK)
					{
						CfgReadStep	= DELETE_DAT_OBJ;
					}
					break;
			}
			break;

		case DELETE_DAT_OBJ:
			DO_Delete.enable	= TRUE;
			DO_Delete.ident		= DO_Info.ident;

			DatObjDelete(&DO_Delete);

			if(DO_Delete.status == ERR_OK)
			{
				CfgReadStep	= CLOSE_MEM_READER;
			}
			break;

		case CLOSE_MEM_READER:
			CloseMemoryReader.enable	= TRUE;
			CloseMemoryReader.ident		= CreateMemoryReader.ident;

			xmlCloseMemoryReader(&CloseMemoryReader);

			if(CloseMemoryReader.status == ERR_OK)
			{
				Start		= FALSE;
				CfgReadStep	= WAIT;
			}
			break;

		case ERROR:
			Start		= FALSE;
			CfgReadStep	= WAIT;
			break;

	}

}

void _EXIT ProgramExit(void)
{

}
```
